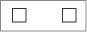
VISUALIZATION VISU_ConfigBOOLEntry_Small  // 87x32
VAR_IN_OUT
    active : BOOL;
    editable : BOOL;
END_VAR
    Checkbox (10,0 45x30), variable: active, input disabled if: TRUE
    Checkbox (60,0 25x30), variable: editable
END_VISUALIZATION

(* stored: Version 1.1.0.1, ProductVersion 3.1.0.36
   Visu VISU_ConfigBOOLEntry_Small: Id {23b135e3-06e1-4967-a37f-9f2f8775f36f} *)
